{attribute 'GeneratedUsingTerminal: EK1100-0000-0018'}
{attribute addProperty BoxType "EK1100-0000-0018"}
{attribute addProperty Id "Beckhoff_EPP4xxxEK1122Beckhoff_EPP4xxxEK1122_FE2E0BEF222"}
{attribute addProperty CRC "4032527010"}
{attribute addProperty Size "222"}
TYPE Beckhoff_EPP4xxx_F05B7AA2 EXTENDS EK1100_1FC0878B :
STRUCT
	{attribute addProperty Name "Beckhoff_EPP4xxxEK1122"}
	{attribute addProperty PreviousPort "Beckhoff EPP4xxx : B"}
	Beckhoff_EPP4xxxEK1122 : Beckhoff_EPP4xxxEK1122_FE2E0BEF;
END_STRUCT
END_TYPE

(* stored: Version 1.2.0.0, ProductVersion 3.1.4024.9
   DUT Beckhoff_EPP4xxx_F05B7AA2: Id {a58ce160-9813-4450-8aee-e9a63a4dcf82} *)
